(* IEC 61131-3 sources: eCockpitGit/test_project/src/%F%02 System/%F%02 Module Manager/%POU%FB_ModuleManager/%F%SYS Module/%PRO%SYS_nameWrite, 1 file *)

(* ---- %GETSET%Get.st ---- *)
VAR
END_VAR

(*%!%__DELIMITER__%!%*)
SYS_nameWrite		:=		TRUE;
